PROGRAM TelescopeAuxiliary
VAR
	MQTTTimer : TON := (PT:=T#5S);
	cycle:	USINT;
	FBReadPressure : FB_ReadAdsSymByName;
	FBReadTemperature: FB_ReadAdsSymByName;
	// EL3064-1
	raw_dewar_pressure		AT%I*: INT;
	pressure_voltage:	REAL;
	dewar_warning_trigger: SR;
	dewar_error_trigger: SR;
	DewarWarning, DewarError: FB_EventLog;
END_VAR
VAR_OUTPUT
	// BT9 mirror
	temperature_mirror2:	REAL;
	// BT10
	temperature_mirror1:	REAL;
	pressure:		REAL;
	temperature:	REAL;
	dewar_pressure:	REAL;
	dewar_pressure_atm: REAL;
END_VAR

temperature_mirror1 := GVL_Telescope.temperature_mirror1 / 1000.0;
temperature_mirror2 := GVL_Telescope.temperature_mirror2 / 1000.0;


cycle := cycle MOD 8;
FBReadPressure(
	bRead := cycle MOD 10 = 1,
	sNetId := '5.40.71.146.1.1',
	sVarName := 'Environment.Pressure',
	nDestAddr := ADR(pressure),
	nLen := SIZEOF(pressure),
 	eComMode := eAdsComModeFastCom
	);
FBReadTemperature(
	bRead := cycle MOD 10 = 4,
	sNetId := '5.40.71.146.1.1',
	sVarName := 'Environment.Temperature1',
	nDestAddr := ADR(temperature),
	nLen := SIZEOF(temperature),
 	eComMode := eAdsComModeFastCom
	);
IF NOT (FBReadPressure.bBusy OR FBReadPressure.bError) AND 
   NOT (FBReadTemperature.bBusy OR FBReadTemperature.bError) THEN
	cycle := cycle + 1;
END_IF

pressure_voltage := F_YREAL(raw_dewar_pressure, 0, 32767, 0.0, 10.0);
dewar_pressure := LREAL_TO_REAL(EXPT(10.0, F_YREAL(pressure_voltage, 2.0, 10.0, -9.0, 3.0)));
dewar_pressure_atm := LREAL_TO_REAL(EXPT(10.0, F_YREAL(pressure_voltage, 2.0, 10.0, -7.0, 5.0)));

dewar_warning_trigger(SET1 := dewar_pressure_atm > 1E-6, RESET := dewar_pressure_atm < 5E-7);
dewar_error_trigger(SET1 := dewar_pressure_atm > 1E-5, RESET := dewar_pressure_atm < 1E-6);

DewarWarning(Trigger := dewar_warning_trigger.Q1,
				Level := ADSLOG_MSGTYPE_WARN,
				FormatString := '%s',
				OnMessage := 'Dewar pressure is above nominal.',
				OffMessage := 'Dewar pressure is nominal.');

DewarWarning(Trigger := dewar_error_trigger.Q1,
				Level := ADSLOG_MSGTYPE_ERROR,
				FormatString := '%s',
				OnMessage := 'Dewar pressure is critical!');

				
MQTTTimer(IN:=TRUE);
IF MQTTTimer.Q THEN // publish new payload every second

	MAIN.MQTTClient.Publish('telescope', 'dome', 'Mirror1Temperature',	LREAL_TO_FMTSTR(temperature_mirror1, 2, TRUE));
	MAIN.MQTTClient.Publish('telescope', 'dome', 'Mirror2Temperature',	LREAL_TO_FMTSTR(temperature_mirror2, 2, TRUE));
	MAIN.MQTTClient.Publish('telescope', 'dome', 'DewarPressureVoltage', LREAL_TO_FMTSTR(pressure_voltage, 3, TRUE));
	MAIN.MQTTClient.Publish('telescope', 'dome', 'DewarPressure', LREAL_TO_FMTSTR(dewar_pressure_atm, 9, TRUE));
	
	MQTTTimer(IN:=FALSE);

END_IF

END_PROGRAM

(* stored: Version 1.1.0.1, ProductVersion 3.1.4024.9
   POU TelescopeAuxiliary: Id {974ce34a-6026-4bc5-b92d-99da70a09948}, SpecialFunc None *)
